(* IEC 61131-3 sources: eCockpitGit/test_project/src/%PLC%PLCTest2/%PLOG%Plc Logic/%APP%APP1_Test/%F%NormalFolder, 5 files *)

(* ---- %DUT%enum_test_1.st ---- *)
{attribute 'qualified_only'}
{attribute 'strict'}
TYPE enum_test_1 :
(
	enum1,
	enum2,
	enum3 := 5
);
END_TYPE

(* ---- %DUT%struct_test_1.st ---- *)
TYPE struct_test_1 :
STRUCT
	structMember1		:BOOL;
	structMember2		:INT;
	structMember3		:STRING;
	structMember4		:WORD;
END_STRUCT
END_TYPE

(* ---- %DUT%union_test_1.st ---- *)
TYPE union_test_1 :
UNION
	union1:BOOL;
	union2:INT;
	union3:WORD;
END_UNION
END_TYPE

(* ---- %POU%fb_test_1.st ---- *)
FUNCTION_BLOCK fb_test_1
VAR_INPUT
END_VAR
VAR_OUTPUT
END_VAR
VAR
END_VAR

(*%!%__DELIMITER__%!%*)

(* ---- %POU%prg_test_1.st ---- *)
PROGRAM prg_test_1
VAR
	testVar1:BOOL;
	testVar2:INT;
	testVar3:STRING;

	alias1		:alias_test;
	enum1		:enum_test;
	struct1		:struct_test;
	union1		:union_test;
END_VAR

(*%!%__DELIMITER__%!%*)
IF testVar1 THEN
	testVar2		:=		44;
END_IF

testVar3[4]			:=		testVar2;
